// TwinCAT 3 PLC project IO
// Title: Inputs and Outputs
// Company: MyCompany
// Author: Sajedeh Taheri
// ProjectVersion: 0.1.0.0
// Description: this library hold functionality for sensors and actuators
// ProgramVersion: 3.1.4024.0
// libraries:
//   Tc2_Standard, * (Beckhoff Automation GmbH)
//   Tc2_System, * (Beckhoff Automation GmbH)
//   Tc3_Module, * (Beckhoff Automation GmbH)
// project tree:
//   / PlcTask.TcTTO (not stored)
//   POUs/ F_factorial.TcPOU (not stored)
//   Version/ Global_Version.TcGVL
// real-time tasks:
//   TASK PlcTask: cycle T#10ms, priority 20, ADS port 350

// ---- Version/Global_Version.TcGVL
{attribute 'TcGenerated'}
{attribute 'no-analysis'}
{attribute 'linkalways'}
// This function has been automatically generated from the project information.
VAR_GLOBAL CONSTANT
	{attribute 'const_non_replaced'}
	stLibVersion_Inputs_and_Outputs : ST_LibVersion := (iMajor := 0, iMinor := 1, iBuild := 0, iRevision := 0, nFlags := 0, sVersion := '0.1.0.0');
END_VAR
